Staubli VAL3: WriteSingleIO.pjx

--- WriteSingleIO.pjx ---
Parameters version=s7.9.1 stackSize=5000 millimeterUnit=true
Program file=start.pgx
Program file=stop.pgx
Data file=WriteSingleIO.dtx

--- WriteSingleIO.dtx ---
public bool bState
public num nModuleId
public num nPin
